KUKA KRL program: chk_w2_wechs_ok.src

&ACCESS RVO3
&REL 5
&COMMENT Check C2
DEF chk_w2_wechs_ok( )

; VERIFICAÇÃO DE FERRAMENTE: C2

WAIT FOR ((($IN[161]) OR ((NOT $IN[161]) AND ($IN [3320]))) AND (not $in[169]) AND (($IN[185]) OR ((NOT $IN[185]) AND ($IN [3320]))) AND ($in[177]) AND ($in[193]) AND ($in[201]) AND ($in[219]))

END
